FUNCTION_BLOCK Win32ErrorCodeDesciption_Tests EXTENDS TcUnit.FB_TestSuite

DescriptionOfKnownErrorCode();
DescriptionOfUnknownErrorCode();

METHOD DescriptionOfKnownErrorCode
TcUnit.TEST('DescriptionOfKnownErrorCode');

AssertEquals_STRING(
    Expected:='The system cannot find the file specified.',
    Actual:=Win32ErrorCodeDescription(Win32ErrorCodes.ERROR_FILE_NOT_FOUND),
    Message:='Error description not correct.'
);

TcUnit.TEST_FINISHED();
END_METHOD

METHOD DescriptionOfUnknownErrorCode
TcUnit.TEST('DescriptionOfUnknownErrorCode');

AssertEquals_STRING(
    Expected:='Unknown Win32 error code.',
    Actual:=Win32ErrorCodeDescription(Win32ErrorCodes.ERR_UNKNOWN),
    Message:='Error description not correct.'
);

TcUnit.TEST_FINISHED();
END_METHOD

END_FUNCTION_BLOCK

(* stored: Version 1.1.0.1, ProductVersion 3.1.4024.11
   POU Win32ErrorCodeDesciption_Tests: Id {2f90ed74-a809-49bb-b887-3ce9960e7cde}, SpecialFunc None
   Method DescriptionOfKnownErrorCode: Id {df328d3c-bff8-450d-8afa-639df839f5ad}
   Method DescriptionOfUnknownErrorCode: Id {da94d620-520f-42ad-a0e2-e07ed6451ef2} *)
